{attribute 'qualified_only'}
{attribute 'strict'}
{attribute 'to_string'}
TYPE E_Chamber1DataId :
(
	None := 0,
	SingleProcess_Prepare_StartUtc := 701,
	SingleProcess_Prepare_EndUtc := 702,
	SingleProcess_Prepare_ActualMs := 703,
	SingleProcess_LiftReady_StartUtc := 704,
	SingleProcess_LiftReady_EndUtc := 705,
	SingleProcess_LiftReady_ActualMs := 706,
	SingleProcess_SpinAlign_StartUtc := 707,
	SingleProcess_SpinAlign_EndUtc := 708,
	SingleProcess_SpinAlign_ActualMs := 709,
	SingleProcess_ConcurrentProcessEntry_StartUtc := 710,
	SingleProcess_ConcurrentProcessEntry_EndUtc := 711,
	SingleProcess_ConcurrentProcessEntry_ActualMs := 712,
	SingleProcess_SpinRampUp_StartUtc := 713,
	SingleProcess_SpinRampUp_EndUtc := 714,
	SingleProcess_SpinRampUp_ActualMs := 715,
	SingleProcess_ProcessHold_StartUtc := 716,
	SingleProcess_ProcessHold_EndUtc := 717,
	SingleProcess_ProcessHold_ActualMs := 718,
	SingleProcess_ConcurrentProcessExit_StartUtc := 719,
	SingleProcess_ConcurrentProcessExit_EndUtc := 720,
	SingleProcess_ConcurrentProcessExit_ActualMs := 721,
	SingleProcess_SpinStandby_StartUtc := 722,
	SingleProcess_SpinStandby_EndUtc := 723,
	SingleProcess_SpinStandby_ActualMs := 724
) UDINT;
END_TYPE

(* stored: Version 1.1.0.1, ProductVersion 3.1.4026.18
   DUT E_Chamber1DataId: Id {8e5229a3-bdb7-4bf6-977a-4bdc96b43819} *)
